# EPICS autosave request: apps/svtIntlkApp/Db/svtIntlk_bpm.req
#
# SVT Soft Interlock settings
#
$(P)intlk_delay
#$(P)intlk_lim
$(P)intlk_bypass
$(P)intlk_reset
$(P)intlk_status
